// Mitsubishi GX Works2 project: e07   PLC: Q02/Q02H

PROGRAM MAIN
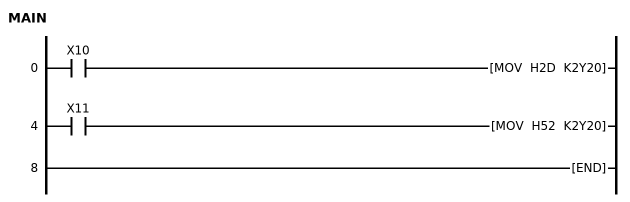
0     LD      X10
      MOV     H2D K2Y20
4     LD      X11
      MOV     H52 K2Y20
8     END
END_PROGRAM
